# B&R Automation Studio project Lab_2
Automation Studio 4.5.2.102

## Configuration Config1

### Task classes (Cpu.sw)
```
Cyclic#1:
  Program <- Program.prg
DataObjects: Acp10sys
NcDataObjects: acp10etxen <- acp10etxen.dob
VcDataObjects: Visu <- Visu.dob
Binaries: udbdef, TCData, arconfig, User, sysconf, iomap, asfw, ashwac, ashwd, Role, acp10cfg, Acp10map
Libraries: Acp10man, Acp10par, NcGlobal, Acp10sdc, AsBrStr, powerlnk, astime, fileio, runtime
```

### Hardware
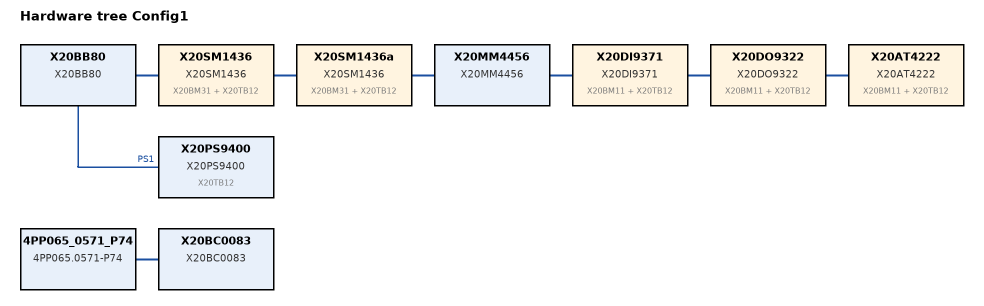
```
4PP065_0571_P74 : 4PP065.0571-P74 v1.1.2.0
  Connector IF5:
    ActivateDevice = 1
    Mode = Manual
    InternetAddress = 127.0.0.1
    SubnetMask = 255.255.255.0
  ConfigurationID = labBR
  Simulation = 1
  TimerDeviceType = EPLX2X
  TimerDevice = 4PP065_0571_P74.IF4
  TaskClassIdleTime = 2000
  Cyclic1Output = 1
  VcObjectName = Visu
X20AT4222 : X20AT4222 v1.2.3.0  [SS1 -> X20TB12e.SS; SL -> X20BM11b.SL1]
X20BB80 : X20BB80 v1.0.2.0
X20BC0083 : X20BC0083 v2.7.0.0  [PLK1 -> 4PP065_0571_P74.IF4 [Cable Type=PowerlinkCable, Length=10, Version=1.0.0.2]; SL -> X20BB80.SL1]
X20BM11 : X20BM11 v1.0.0.1  [X2X1 -> X20MM4456.X2X2]
X20BM11a : X20BM11 v1.0.0.1  [X2X1 -> X20BM11.X2X2]
X20BM11b : X20BM11 v1.0.0.1  [X2X1 -> X20BM11a.X2X2]
X20BM31 : X20BM31 v1.0.0.1  [X2X1 -> X20BB80.IF1]
X20BM31a : X20BM31 v1.0.0.1  [X2X1 -> X20BM31.X2X2]
X20DI9371 : X20DI9371 v1.0.2.0  [SS1 -> X20TB12c.SS; SL -> X20BM11.SL1]
X20DO9322 : X20DO9322 v1.0.3.0  [SS1 -> X20TB12d.SS; SL -> X20BM11a.SL1]
X20MM4456 : X20MM4456 v1.1.5.0  [X2X1 -> X20BM31a.X2X2]
X20PS9400 : X20PS9400 v1.0.2.4  [SS1 -> X20TB12.SS; PS -> X20BB80.PS1]
X20SM1436 : X20SM1436 v1.4.2.1  [SS1 -> X20TB12a.SS; SL -> X20BM31.SL1]
X20SM1436a : X20SM1436 v1.4.2.1  [SS1 -> X20TB12b.SS; SL -> X20BM31a.SL1]
X20TB12 : X20TB12 v1.0.0.0
X20TB12a : X20TB12 v1.0.0.0
X20TB12b : X20TB12 v1.0.0.0
X20TB12c : X20TB12 v1.0.0.0
X20TB12d : X20TB12 v1.0.0.0
X20TB12e : X20TB12 v1.0.0.0
```

## Logical view

### Program Logical/Program (ANSIC)

#### Variables.var
```iecst
VAR
	LED : ARRAY[0..3] OF BOOL := [3(1),0];
	BTN : ARRAY[0..3] OF BOOL := [4(0)];
END_VAR
```

#### Main.c
```c
#include <bur/plctypes.h>

#ifdef _DEFAULT_INCLUDES
#include <AsDefault.h>
#endif

void _INIT ProgramInit(void) {

}

void _CYCLIC ProgramCyclic(void) {
	LED[0] = 1;
	LED[1] = 1;
	LED[2] = 1;
	LED[3] = 0;

	if (BTN[0]) {
		LED[1] = !LED[1];
	}
	if (BTN[1]) {
		LED[0] = !LED[0];
		LED[1] = !LED[1];
		LED[3] = !LED[3];
	}
	if (BTN[2]) {
		LED[0] = !LED[0];
		LED[2] = !LED[2];
	}
	if (BTN[4]) {
		LED[0] = !LED[0];
		LED[2] = !LED[2];
		LED[3] = !LED[3];
	}
}

void _EXIT ProgramExit(void) {

}
```

- Visualisation Logical/Visu (not shown)

Listed in the project but not available here: Logical/Global.typ, Logical/Global.var, Logical/Libraries, Logical/acp10etxen
